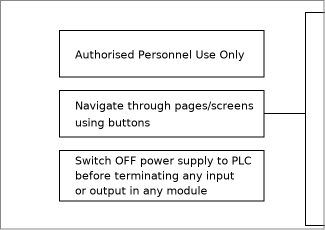
VISUALIZATION V_Main  // 325x230
    Rectangle (59,150 205x51)
    Rectangle (59,90 205x47)
    Rectangle (59,30 205x47)
    Label (72,98 185x21), "Navigate through pages/screens"
    Label (72,153 191x31), "Switch OFF power supply to PLC"
    Label (72,168 181x31), "before terminating any input"
    Label (72,47 183x21), "Authorised Personnel Use Only"
    Line (305,12) (305,225)
    Line (264,113) (305,113)
    Line (305,12) (325,12)
    Line (305,225) (325,225)
    Label (72,115 177x21), "using buttons"
    Label (72,183 146x20), "or output in any module"
END_VISUALIZATION

(* stored: Version 1.1.0.1, ProductVersion 3.1.4024.11
   Visu V_Main: Id {a9e1b69a-b223-4288-bc89-92b58396e565} *)
